(*			
	RafalOS
	Rafał Osajda		20.11.2025		TC 4024.66
	Moduł przygotowania danych dla Okna statystyk we wszsytkich trybach
*)
FUNCTION_BLOCK FB_MCHMIPrepareDataForScreen_05_XX EXTENDS FB_MCHMIPrepareDataForScreen IMPLEMENTS ITF_MCHMIPrepareDataForScreen
VAR
	itfMachineControlHMI	: ITF_MCHMIMachineControl_HMI_PrepScr_05_XX;
	refstData				: REFERENCE TO ST_MCHMIPrepareScreen_05_XX;
END_VAR

(*			
	RafalOS
	Rafał Osajda		19.11.2025		TC 4024.66
	Czyści danych przy zmienia ramki po poprzedniej ramce
*)
METHOD PUBLIC ClearAfterScreen : BOOL
VAR_INPUT
END_VAR
SUPER^.ClearAfterScreen ();
END_METHOD

METHOD PUBLIC LinkDataHMI_05_XX : BOOL
VAR_INPUT
	refstData				: REFERENCE TO ST_MCHMIPrepareScreen_05_XX;
END_VAR
THIS^.refstData REF= refstData;
END_METHOD

METHOD PUBLIC LinkMachineControlHMI : BOOL
VAR_INPUT
	fbMachineControlHMI	: ITF_MCHMIMachineControl_HMI_PrepScr_05_XX;
END_VAR
this^.itfMachineControlHMI := fbMachineControlHMI;
END_METHOD

(*			
	RafalOS
	Rafał Osajda		14.11.2025		TC 4024.66
	Metoda przygotowywania danych dla HMI 
	W niej odbywa się odpytywanie właściego elementu przez łącznik
*)
METHOD PUBLIC PrepareDataForHMI : BOOL
VAR_INPUT
END_VAR
SUPER^.PrepareDataForHMI ();
END_METHOD

(*			
	RafalOS
	Rafał Osajda		19.11.2025		TC 4024.66
	Przygotowanie ramki pood tamke do wyświetlenia - tylko przygotowanie a nie przygotowanie danych do wyświetlenia
*)
METHOD PUBLIC PrepareForScreen : BOOL
VAR_INPUT
END_VAR
SUPER^.PrepareForScreen ();
END_METHOD

END_FUNCTION_BLOCK

(* stored: Version 1.1.0.1
   POU FB_MCHMIPrepareDataForScreen_05_XX: Id {ac3c59d3-431d-07ad-150f-33041e514b62}, SpecialFunc None
   Folder ITF_PDFS: Id {a75f3db2-688d-0ec4-2718-d01bc83acdd2}
   Method ClearAfterScreen: Id {9408c0e3-1816-0bda-38aa-142e6b23d2c5}
   Method LinkDataHMI_05_XX: Id {c527c097-b7d4-07eb-0e82-69d343bae913}
   Method LinkMachineControlHMI: Id {93bf0eda-f251-04cc-3674-0f3fcd416897}
   Method PrepareDataForHMI: Id {29f88666-dbfb-07fb-14f7-d297ff97679e}
   Method PrepareForScreen: Id {98d5a362-da4d-071c-21b5-143c2384a935} *)
